// TIA Portal project "FinalYearProjectCode" (V17)
// This is the final combined plc code for the 5th year project

(* hardware
DEVICE "S7-1200 station_1"  S7-1200 Station
   slot 0: "Rack_0"  S7-1200 Rack  Rack  V1.0
   slot 1: "PLC_1"  CPU 1214C DC/DC/DC  6ES7 214-1AG40-0XB0  V4.2
   slot 2: "AI 4x13BIT/AQ 2x14BIT_1"  6ES7 234-4HE32-0XB0  V2.1
DEVICE "HMI_1"  TP700 Comfort
   slot 0: "HMI_1"  TP700 Comfort  6AV2 124-0GC01-0AX0  17.0.0.0
   slot 1: "HMI_RT_1"  TP700 Comfort  6AV2 124-0GC01-0AX0  17.0.0.0
   slot 5: "HMI_1.IE_CP_1"  PROFINET Interface  17.0.0.0
      slot 1: "PROFINET Interface_1"  PROFINET Interface
         slot 1: "Port_1"  Port
         slot 2: "Port_2"  Port
   slot 7: "HMI_1.MPI/DP_CP_1"  MPI/DP Interface  17.0.0.0
*)

// ===== PLC "PLC_1"  CPU 1214C DC/DC/DC =====

VAR_GLOBAL   // PLC tag table "Default tag table"
   "System_Byte" AT %MB100 : Byte;
   "FirstScan" AT %M100.0 : Bool;
   "DiagStatusUpdate" AT %M100.1 : Bool;
   "AlwaysTRUE" AT %M100.2 : Bool;
   "AlwaysFALSE" AT %M100.3 : Bool;
   "Clock_Byte" AT %MB101 : Byte;
   "Clock_10Hz" AT %M101.0 : Bool;
   "Clock_5Hz" AT %M101.1 : Bool;
   "Clock_2.5Hz" AT %M101.2 : Bool;
   "Clock_2Hz" AT %M101.3 : Bool;
   "Clock_1.25Hz" AT %M101.4 : Bool;
   "Clock_1Hz" AT %M101.5 : Bool;
   "Clock_0.625Hz" AT %M101.6 : Bool;
   "Clock_0.5Hz" AT %M101.7 : Bool;
END_VAR

VAR_GLOBAL   // PLC tag table "i_o_tags"
   "Voltage_transmitter" AT %IW96 : Int;
   "i_p_transducer" AT %QW96 : Int;
   "solar_sync" AT %Q0.1 : Bool;
   "compressor_rel" AT %Q0.2 : Bool;
   "caes_sync" AT %Q0.3 : Bool;
END_VAR

VAR_GLOBAL   // PLC tag table "HMI_tags"
   "HMI_START" AT %M0.0 : Bool;
   "HMI_STOP" AT %M0.1 : Bool;
   "Current_mode" AT %M0.2 : Bool;
END_VAR

VAR_GLOBAL   // PLC tag table "outMem_tags"
   "solarMainSync" AT %M1.0 : Bool;
   "solarStartSync" AT %M1.1 : Bool;
   "solarOnlySync" AT %M1.2 : Bool;
END_VAR

VAR_GLOBAL   // PLC tag table "caes_tags"
   "freq_feedback" AT %MD10 : Real;
   "first_in" AT %MD14 : Real;
   "i_p_mem1" AT %MW18 : Int;
   "controller_output" AT %MD20 : Real;
   "feedback_scale" AT %MD24 : Real;
   "control_scale" AT %MD28 : Real;
   "i_p_mem_2" AT %MW32 : Int;
   "press_mem" AT %MD34 : Real;
   "HMI_pressure" AT %MD38 : Real;
   "caesControlError" AT %MD42 : Real;
END_VAR

DATA_BLOCK "modbusConfig"   // DB3
{ S7_Optimized_Access := 'TRUE' }
VERSION : 0.1
   VAR
      MB_MODE : USInt;
      MB_DATA_ADDR_1 : UDInt := 30051;
      MB_DATA_ADDR_2 : UDInt := 30061;
      MB_DATA_ADDR_3 : UDInt := 30071;
      MB_DATA_ADDR_4 : UDInt := 30081;
      MB_DATA_ADDR_5 : UDInt := 30091;
      MB_DATA_LEN : UInt := 1;
      CONNECT_1 : TCON_IP_v4;
      CONNECT_2 : TCON_IP_v4;
      CONNECT_3 : TCON_IP_v4;
      CONNECT_4 : TCON_IP_v4;
      CONNECT_5 : TCON_IP_v4;
      STATUS_1 : Word;
      STATUS_2 : Word;
      STATUS_3 : Word;
      STATUS_4 : Word;
      STATUS_5 : Word;
      ERROR_1 : Bool;
      ERROR_2 : Bool;
      ERROR_3 : Bool;
      ERROR_4 : Bool;
      ERROR_5 : Bool;
   END_VAR
BEGIN
   CONNECT_1.InterfaceId := 64;
   CONNECT_1.ID := 1;
   CONNECT_1.ActiveEstablished := true;
   CONNECT_1.RemoteAddress.ADDR[1] := 172;
   CONNECT_1.RemoteAddress.ADDR[2] := 16;
   CONNECT_1.RemoteAddress.ADDR[3] := 41;
   CONNECT_1.RemoteAddress.ADDR[4] := 240;
   CONNECT_1.RemotePort := 502;
   CONNECT_2.InterfaceId := 64;
   CONNECT_2.ID := 2;
   CONNECT_2.ActiveEstablished := true;
   CONNECT_2.RemoteAddress.ADDR[1] := 172;
   CONNECT_2.RemoteAddress.ADDR[2] := 16;
   CONNECT_2.RemoteAddress.ADDR[3] := 41;
   CONNECT_2.RemoteAddress.ADDR[4] := 240;
   CONNECT_2.RemotePort := 502;
   CONNECT_3.InterfaceId := 64;
   CONNECT_3.ID := 3;
   CONNECT_3.ActiveEstablished := true;
   CONNECT_3.RemoteAddress.ADDR[1] := 172;
   CONNECT_3.RemoteAddress.ADDR[2] := 16;
   CONNECT_3.RemoteAddress.ADDR[3] := 41;
   CONNECT_3.RemoteAddress.ADDR[4] := 240;
   CONNECT_3.RemotePort := 502;
   CONNECT_4.InterfaceId := 64;
   CONNECT_4.ID := 4;
   CONNECT_4.ActiveEstablished := true;
   CONNECT_4.RemoteAddress.ADDR[1] := 172;
   CONNECT_4.RemoteAddress.ADDR[2] := 16;
   CONNECT_4.RemoteAddress.ADDR[3] := 41;
   CONNECT_4.RemoteAddress.ADDR[4] := 240;
   CONNECT_4.RemotePort := 502;
   CONNECT_5.InterfaceId := 64;
   CONNECT_5.ID := 5;
   CONNECT_5.ActiveEstablished := true;
   CONNECT_5.RemotePort := 502;
   CONNECT_5.RemoteAddress.ADDR[1] := 172;
   CONNECT_5.RemoteAddress.ADDR[2] := 16;
   CONNECT_5.RemoteAddress.ADDR[3] := 41;
   CONNECT_5.RemoteAddress.ADDR[4] := 240;
END_DATA_BLOCK

DATA_BLOCK "mbDataPTR"   // DB4
{ S7_Optimized_Access := 'FALSE' }
VERSION : 0.1
   VAR
      loadCurrent : Word;
      mainBusFreq : Word;
      solarSync : Word;
      solarFailsafe : Word;
      caesFailSafe : Word;
   END_VAR
BEGIN
END_DATA_BLOCK

FUNCTION "CAESControl" : Void   // FC1, LAD
{ S7_Optimized_Access := 'TRUE' }
VERSION : 0.1
BEGIN

REGION Network 1: Generator start_up
   // This block sets the generator
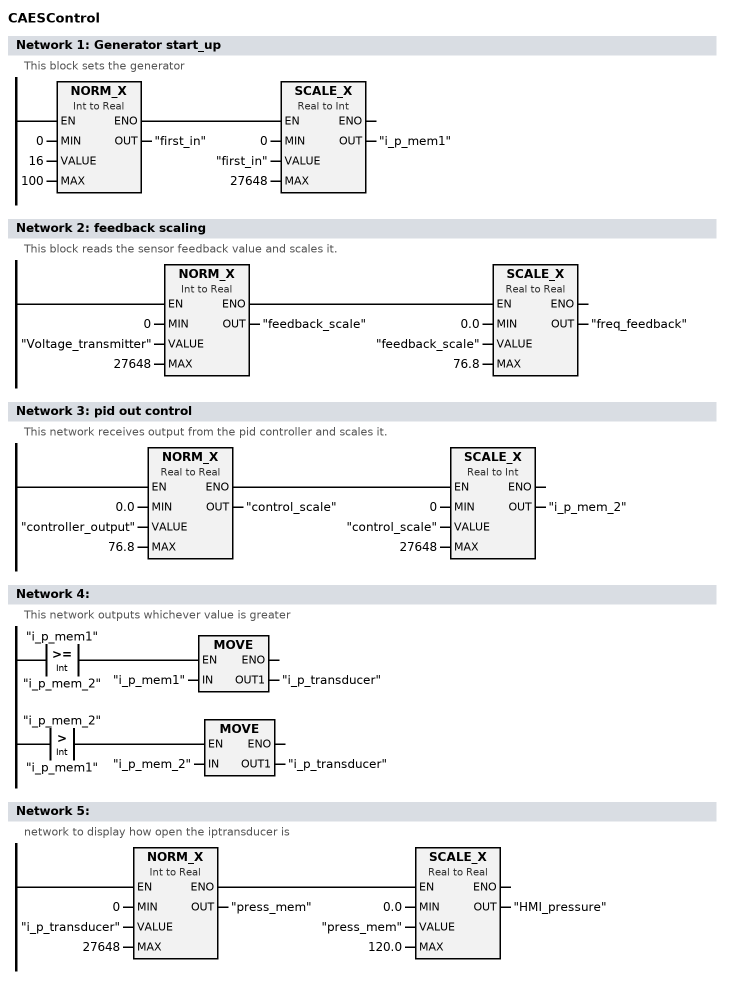
   RUNG wire#powerrail
      { S7_Templates := "[SrcType := Int, DestType := Real]" } Normalize(min := 0, value := 16, max := 100, out => "first_in")
      { S7_Templates := "[SrcType := Real, DestType := Int]" } Scale(min := 0, value := "first_in", max := 27648, out => "i_p_mem1")
   END_RUNG
   // the same network as SCL:
   "first_in" := NORM_X(MIN := 0, VALUE := 16, MAX := 100);
   "i_p_mem1" := SCALE_X(MIN := 0, VALUE := "first_in", MAX := 27648);
END_REGION

REGION Network 2: feedback scaling
   // This block reads the sensor feedback value and scales it.
   RUNG wire#powerrail
      { S7_Templates := "[SrcType := Int, DestType := Real]" } Normalize(min := 0, value := "Voltage_transmitter", max := 27648, out => "feedback_scale")
      { S7_Templates := "[SrcType := Real, DestType := Real]" } Scale(min := 0.0, value := "feedback_scale", max := 76.8, out => "freq_feedback")
   END_RUNG
   // the same network as SCL:
   "feedback_scale" := NORM_X(MIN := 0, VALUE := "Voltage_transmitter", MAX := 27648);
   "freq_feedback" := SCALE_X(MIN := 0.0, VALUE := "feedback_scale", MAX := 76.8);
END_REGION

REGION Network 3: pid out control
   // This network receives output from the pid controller and scales it.
   RUNG wire#powerrail
      { S7_Templates := "[SrcType := Real, DestType := Real]" } Normalize(min := 0.0, value := "controller_output", max := 76.8, out => "control_scale")
      { S7_Templates := "[SrcType := Real, DestType := Int]" } Scale(min := 0, value := "control_scale", max := 27648, out => "i_p_mem_2")
   END_RUNG
   // the same network as SCL:
   "control_scale" := NORM_X(MIN := 0.0, VALUE := "controller_output", MAX := 76.8);
   "i_p_mem_2" := SCALE_X(MIN := 0, VALUE := "control_scale", MAX := 27648);
END_REGION

REGION Network 4
   // This network outputs whichever value is greater
   RUNG wire#powerrail
      { S7_Templates := "SrcType := Int" } GE_Contact(in1 := "i_p_mem1", in2 := "i_p_mem_2")
      Move(in := "i_p_mem1", out1 => "i_p_transducer")
   END_RUNG
   RUNG wire#powerrail
      { S7_Templates := "SrcType := Int" } GT_Contact(in1 := "i_p_mem_2", in2 := "i_p_mem1")
      Move(in := "i_p_mem_2", out1 => "i_p_transducer")
   END_RUNG
   // the same network as SCL:
   IF "i_p_mem1" >= "i_p_mem_2" THEN "i_p_transducer" := "i_p_mem1"; END_IF;
   IF "i_p_mem_2" > "i_p_mem1" THEN "i_p_transducer" := "i_p_mem_2"; END_IF;
END_REGION

REGION Network 5
   // network to display how open the iptransducer is
   RUNG wire#powerrail
      { S7_Templates := "[SrcType := Int, DestType := Real]" } Normalize(min := 0, value := "i_p_transducer", max := 27648, out => "press_mem")
      { S7_Templates := "[SrcType := Real, DestType := Real]" } Scale(min := 0.0, value := "press_mem", max := 120.0, out => "HMI_pressure")
   END_RUNG
   // the same network as SCL:
   "press_mem" := NORM_X(MIN := 0, VALUE := "i_p_transducer", MAX := 27648);
   "HMI_pressure" := SCALE_X(MIN := 0.0, VALUE := "press_mem", MAX := 120.0);
END_REGION
END_FUNCTION

FUNCTION "comm" : Void   // FC2, LAD
{ S7_Optimized_Access := 'TRUE' }
VERSION : 0.1
BEGIN

REGION Network 1: Receive Load current
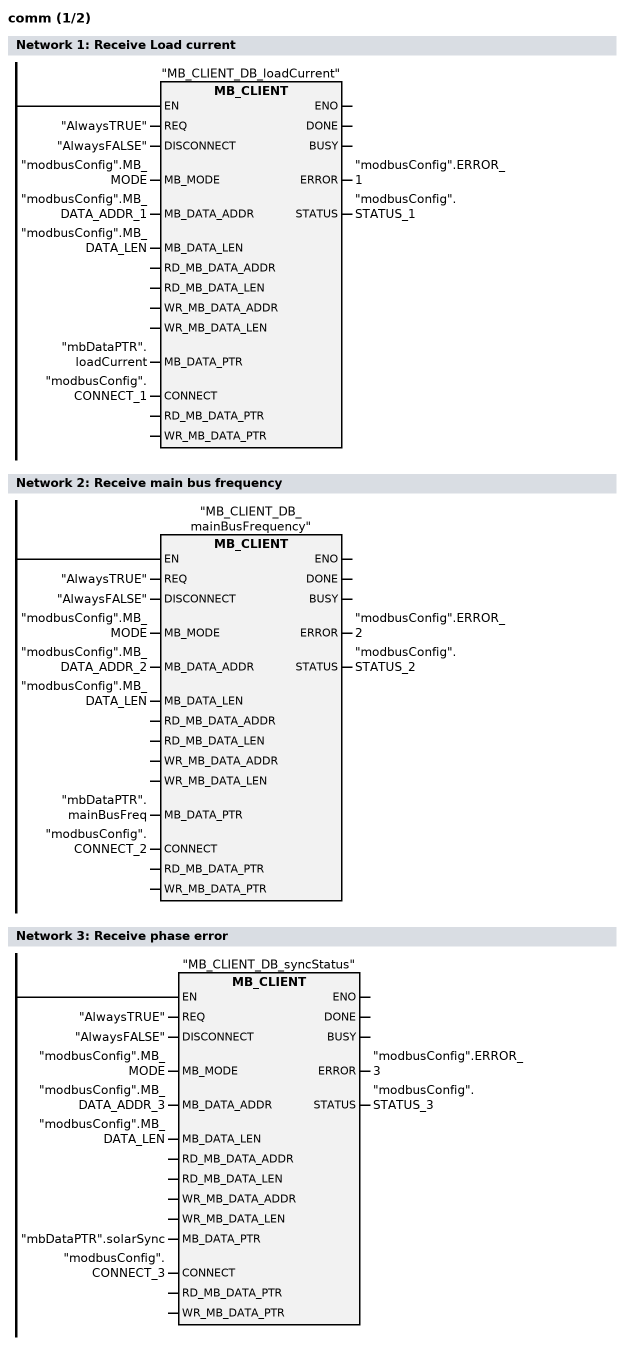
   "MB_CLIENT_DB_loadCurrent"(REQ := "AlwaysTRUE",   // MB_CLIENT
                           DISCONNECT := "AlwaysFALSE",
                           MB_MODE := "modbusConfig".MB_MODE,
                           MB_DATA_ADDR := "modbusConfig".MB_DATA_ADDR_1,
                           MB_DATA_LEN := "modbusConfig".MB_DATA_LEN,
                           MB_DATA_PTR := "mbDataPTR".loadCurrent,
                           CONNECT := "modbusConfig".CONNECT_1,
                           ERROR => "modbusConfig".ERROR_1,
                           STATUS => "modbusConfig".STATUS_1);
END_REGION

REGION Network 2: Receive main bus frequency
   "MB_CLIENT_DB_mainBusFrequency"(REQ := "AlwaysTRUE",   // MB_CLIENT
                           DISCONNECT := "AlwaysFALSE",
                           MB_MODE := "modbusConfig".MB_MODE,
                           MB_DATA_ADDR := "modbusConfig".MB_DATA_ADDR_2,
                           MB_DATA_LEN := "modbusConfig".MB_DATA_LEN,
                           MB_DATA_PTR := "mbDataPTR".mainBusFreq,
                           CONNECT := "modbusConfig".CONNECT_2,
                           ERROR => "modbusConfig".ERROR_2,
                           STATUS => "modbusConfig".STATUS_2);
END_REGION

REGION Network 3: Receive phase error
   "MB_CLIENT_DB_syncStatus"(REQ := "AlwaysTRUE",   // MB_CLIENT
                           DISCONNECT := "AlwaysFALSE",
                           MB_MODE := "modbusConfig".MB_MODE,
                           MB_DATA_ADDR := "modbusConfig".MB_DATA_ADDR_3,
                           MB_DATA_LEN := "modbusConfig".MB_DATA_LEN,
                           MB_DATA_PTR := "mbDataPTR".solarSync,
                           CONNECT := "modbusConfig".CONNECT_3,
                           ERROR => "modbusConfig".ERROR_3,
                           STATUS => "modbusConfig".STATUS_3);
END_REGION

REGION Network 4: Receive CAES Failsafe
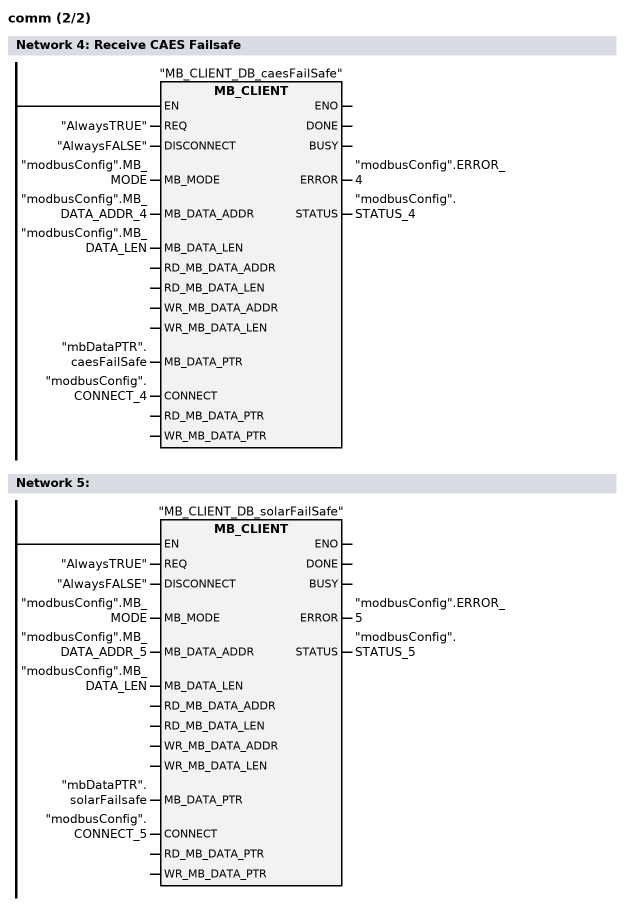
   "MB_CLIENT_DB_caesFailSafe"(REQ := "AlwaysTRUE",   // MB_CLIENT
                           DISCONNECT := "AlwaysFALSE",
                           MB_MODE := "modbusConfig".MB_MODE,
                           MB_DATA_ADDR := "modbusConfig".MB_DATA_ADDR_4,
                           MB_DATA_LEN := "modbusConfig".MB_DATA_LEN,
                           MB_DATA_PTR := "mbDataPTR".caesFailSafe,
                           CONNECT := "modbusConfig".CONNECT_4,
                           ERROR => "modbusConfig".ERROR_4,
                           STATUS => "modbusConfig".STATUS_4);
END_REGION

REGION Network 5
   "MB_CLIENT_DB_solarFailSafe"(REQ := "AlwaysTRUE",   // MB_CLIENT
                           DISCONNECT := "AlwaysFALSE",
                           MB_MODE := "modbusConfig".MB_MODE,
                           MB_DATA_ADDR := "modbusConfig".MB_DATA_ADDR_5,
                           MB_DATA_LEN := "modbusConfig".MB_DATA_LEN,
                           MB_DATA_PTR := "mbDataPTR".solarFailsafe,
                           CONNECT := "modbusConfig".CONNECT_5,
                           ERROR => "modbusConfig".ERROR_5,
                           STATUS => "modbusConfig".STATUS_5);
END_REGION
END_FUNCTION

FUNCTION "StopMode" : Void   // FC3, LAD
{ S7_Optimized_Access := 'TRUE' }
VERSION : 0.1
BEGIN

REGION Network 1
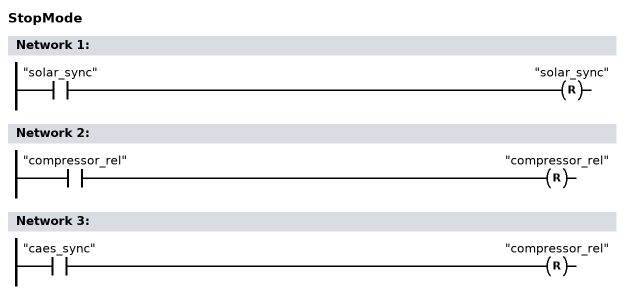
   RUNG wire#powerrail
      Contact( "solar_sync" )
      R_Coil( "solar_sync" )
   END_RUNG
   // the same network as SCL:
   IF "solar_sync" THEN "solar_sync" := FALSE; END_IF;
END_REGION

REGION Network 2
   RUNG wire#powerrail
      Contact( "compressor_rel" )
      R_Coil( "compressor_rel" )
   END_RUNG
   // the same network as SCL:
   IF "compressor_rel" THEN "compressor_rel" := FALSE; END_IF;
END_REGION

REGION Network 3
   RUNG wire#powerrail
      Contact( "caes_sync" )
      R_Coil( "compressor_rel" )
   END_RUNG
   // the same network as SCL:
   IF "caes_sync" THEN "compressor_rel" := FALSE; END_IF;
END_REGION
END_FUNCTION

FUNCTION "runMode" : Void   // FC4, LAD
{ S7_Optimized_Access := 'TRUE' }
VERSION : 0.1
BEGIN

REGION Network 1
   // This network controls the compressor socket
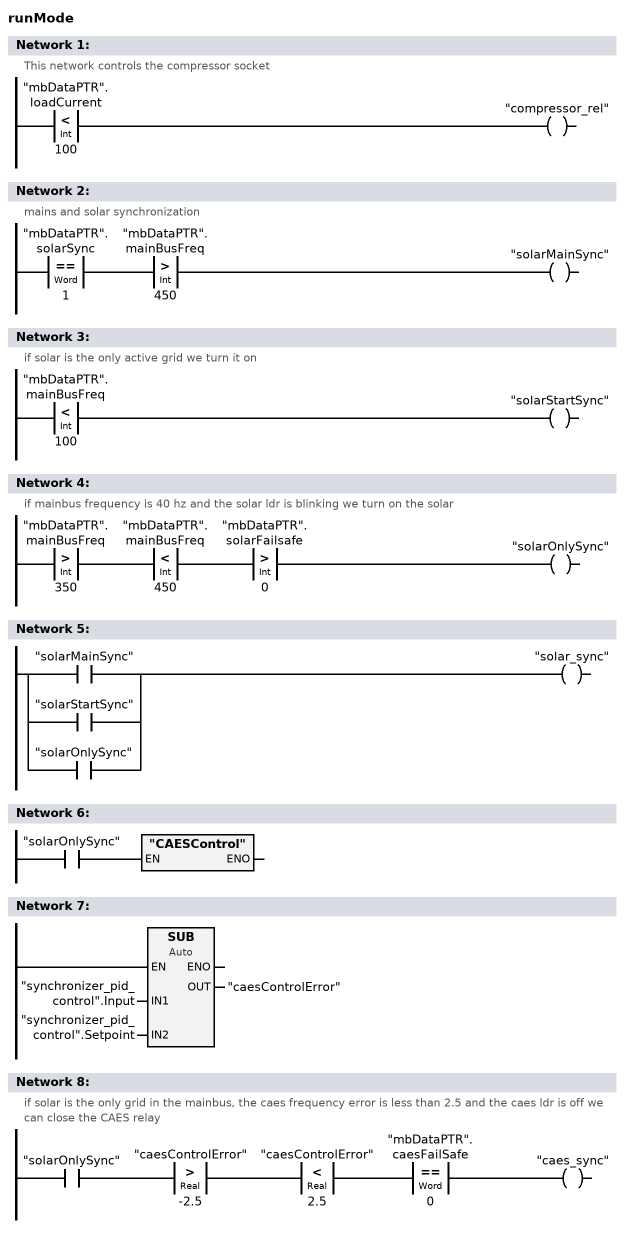
   RUNG wire#powerrail
      { S7_Templates := "SrcType := Int" } LT_Contact(in1 := "mbDataPTR".loadCurrent, in2 := 100)
      Coil( "compressor_rel" )
   END_RUNG
   // the same network as SCL:
   "compressor_rel" := "mbDataPTR".loadCurrent < 100;
END_REGION

REGION Network 2
   // mains and solar synchronization
   RUNG wire#powerrail
      { S7_Templates := "SrcType := Word" } EQ_Contact(in1 := "mbDataPTR".solarSync, in2 := 1)
      { S7_Templates := "SrcType := Int" } GT_Contact(in1 := "mbDataPTR".mainBusFreq, in2 := 450)
      Coil( "solarMainSync" )
   END_RUNG
   // the same network as SCL:
   "solarMainSync" := ("mbDataPTR".solarSync = 1) AND ("mbDataPTR".mainBusFreq > 450);
END_REGION

REGION Network 3
   // if solar is the only active grid we turn it on
   RUNG wire#powerrail
      { S7_Templates := "SrcType := Int" } LT_Contact(in1 := "mbDataPTR".mainBusFreq, in2 := 100)
      Coil( "solarStartSync" )
   END_RUNG
   // the same network as SCL:
   "solarStartSync" := "mbDataPTR".mainBusFreq < 100;
END_REGION

REGION Network 4
   // if mainbus frequency is 40 hz and the solar ldr is blinking we turn on the solar
   RUNG wire#powerrail
      { S7_Templates := "SrcType := Int" } GT_Contact(in1 := "mbDataPTR".mainBusFreq, in2 := 350)
      { S7_Templates := "SrcType := Int" } LT_Contact(in1 := "mbDataPTR".mainBusFreq, in2 := 450)
      { S7_Templates := "SrcType := Int" } GT_Contact(in1 := "mbDataPTR".solarFailsafe, in2 := 0)
      Coil( "solarOnlySync" )
   END_RUNG
   // the same network as SCL:
   "solarOnlySync" := ("mbDataPTR".mainBusFreq > 350) AND ("mbDataPTR".mainBusFreq < 450) AND ("mbDataPTR".solarFailsafe > 0);
END_REGION

REGION Network 5
   RUNG wire#powerrail
      Contact( "solarMainSync" )
      wire#w1
      Coil( "solar_sync" )
   END_RUNG
   RUNG wire#powerrail
      Contact( "solarStartSync" )
   END_RUNG wire#w1
   RUNG wire#powerrail
      Contact( "solarOnlySync" )
   END_RUNG wire#w1
   // the same network as SCL:
   "solar_sync" := "solarMainSync" OR "solarStartSync" OR "solarOnlySync";
END_REGION

REGION Network 6
   RUNG wire#powerrail
      Contact( "solarOnlySync" )
      "CAESControl"()
   END_RUNG
   // the same network as SCL:
   IF "solarOnlySync" THEN "CAESControl"(); END_IF;
END_REGION

REGION Network 7
   RUNG wire#powerrail
      Sub(in1 := "synchronizer_pid_control".Input, in2 := "synchronizer_pid_control".Setpoint, out => "caesControlError")
   END_RUNG
   // the same network as SCL:
   "caesControlError" := "synchronizer_pid_control".Input - "synchronizer_pid_control".Setpoint;
END_REGION

REGION Network 8
   // if solar is the only grid in the mainbus, the caes frequency error is less than 2.5 and the caes ldr is off we can close the CAES relay
   RUNG wire#powerrail
      Contact( "solarOnlySync" )
      { S7_Templates := "SrcType := Real" } GT_Contact(in1 := "caesControlError", in2 := -2.5)
      { S7_Templates := "SrcType := Real" } LT_Contact(in1 := "caesControlError", in2 := 2.5)
      { S7_Templates := "SrcType := Word" } EQ_Contact(in1 := "mbDataPTR".caesFailSafe, in2 := 0)
      Coil( "caes_sync" )
   END_RUNG
   // the same network as SCL:
   "caes_sync" := "solarOnlySync" AND ("caesControlError" > (-2.5)) AND ("caesControlError" < 2.5) AND ("mbDataPTR".caesFailSafe = 0);
END_REGION
END_FUNCTION

ORGANIZATION_BLOCK "Main"   // OB1, LAD, ProgramCycle
TITLE = "Main Program Sweep (Cycle)"
{ S7_Optimized_Access := 'TRUE' }
VERSION : 0.1
   VAR_INPUT
      Initial_Call : Bool;   // Initial call of this OB
      Remanence : Bool;   // =True, if remanent data are available
   END_VAR
BEGIN

REGION Network 1
   // this calls the CAES control circuit
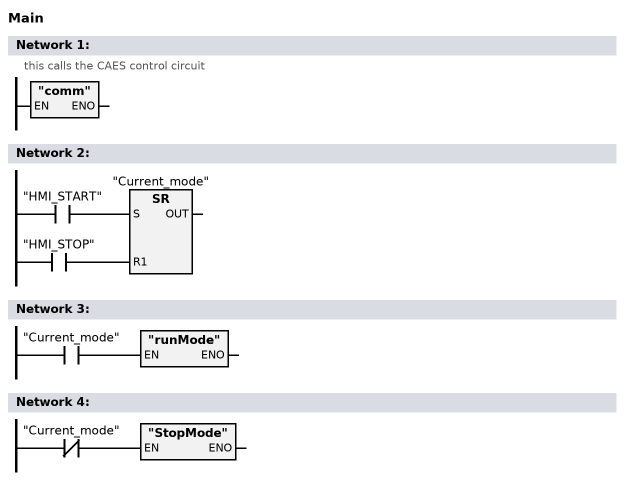
   RUNG wire#powerrail
      "comm"()
   END_RUNG
   // the same network as SCL:
   "comm"();
END_REGION

REGION Network 2
   RUNG wire#powerrail
      Contact( "HMI_START" )
      S_SR(operand := "Current_mode", r1 := wire#w1)
   END_RUNG
   RUNG wire#powerrail
      Contact( "HMI_STOP" )
   END_RUNG wire#w1
   // the same network as SCL:
   IF "HMI_START" THEN
       "Current_mode" := TRUE;   // SR flip-flop
   END_IF;
   IF "HMI_STOP" THEN "Current_mode" := FALSE; END_IF;
END_REGION

REGION Network 3
   RUNG wire#powerrail
      Contact( "Current_mode" )
      "runMode"()
   END_RUNG
   // the same network as SCL:
   IF "Current_mode" THEN "runMode"(); END_IF;
END_REGION

REGION Network 4
   RUNG wire#powerrail
      I_Contact( "Current_mode" )
      "StopMode"()
   END_RUNG
   // the same network as SCL:
   IF NOT "Current_mode" THEN "StopMode"(); END_IF;
END_REGION
END_ORGANIZATION_BLOCK

ORGANIZATION_BLOCK "Cyclic interrupt"   // OB30, LAD, CyclicInterrupt
{ S7_Optimized_Access := 'TRUE' }
VERSION : 0.1
   VAR_INPUT
      Initial_Call : Bool;   // Initial call of this OB
      Event_Count : Int;   // Events discarded
   END_VAR
BEGIN

REGION Network 1
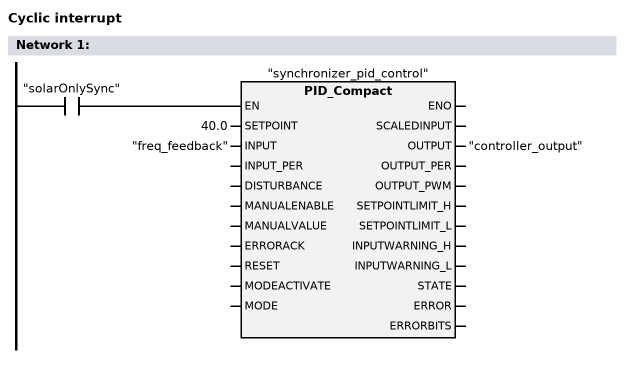
   IF "solarOnlySync" THEN
       "synchronizer_pid_control"(Setpoint := 40.0, Input := "freq_feedback", Output => "controller_output");   // PID_Compact
   END_IF;
END_REGION
END_ORGANIZATION_BLOCK

(* ===== HMI "HMI_RT_1" =====
system functions are stored by id; their names below are inferred from use
connection "HMI_Connection_1": ETHERNET, S7_1200_OMS

HMI tags "Default tag table"
   "synchronizer_pid_control_Output" : Real = PLC synchronizer_pid_control.Output, 1 s
   "synchronizer_pid_control_Input" : Real = PLC synchronizer_pid_control.Input, 1 s
   "synchronizer_pid_control_Setpoint" : Real = PLC synchronizer_pid_control.Setpoint, 1 s
   "synchronizer_pid_control_CtrlParamsBackUp_Gain" : Real = PLC synchronizer_pid_control.CtrlParamsBackUp.Gain, 1 s
   "synchronizer_pid_control_CtrlParamsBackUp_Ti" : Real = PLC synchronizer_pid_control.CtrlParamsBackUp.Ti, 1 s
   "synchronizer_pid_control_CtrlParamsBackUp_Td" : Real = PLC synchronizer_pid_control.CtrlParamsBackUp.Td, 1 s
   "HMI_pressure" : Real = PLC HMI_pressure AT %MD38, 1 s
   "mbDataPTR_loadCurrent" : Word = PLC mbDataPTR.loadCurrent AT %DB4.DBW0, 1 s
   "mbDataPTR_mainBusFreq" : Word = PLC mbDataPTR.mainBusFreq AT %DB4.DBW2, 1 s
   "mbDataPTR_solarSync" : Word = PLC mbDataPTR.solarSync AT %DB4.DBW4, 1 s
   "mbDataPTR_caesFailSafe" : Word = PLC mbDataPTR.caesFailSafe AT %DB4.DBW8, 1 s
   "mbDataPTR_solarFailsafe" : Word = PLC mbDataPTR.solarFailsafe AT %DB4.DBW6, 1 s
   "HMI_START" : Bool = PLC HMI_START AT %M0.0, 1 s
   "HMI_STOP" : Bool = PLC HMI_STOP AT %M0.1, 1 s

screen "CAES_PID" 800x480
   TrendView "Trend view_1" at 3,41 size 594x437
   TextField "Text field_1" at 151,8 size 543x34; Text 'CAES PID CONTROLLER VISUALIZATION'
   IOField "I/O field_1" at 699,43 size 96x32; FormatPattern 99.999
      ProcessValue <- "synchronizer_pid_control_CtrlParamsBackUp_Gain"
   IOField "I/O field_2" at 700,86 size 96x32; FormatPattern 99.999
      ProcessValue <- "synchronizer_pid_control_CtrlParamsBackUp_Ti"
   IOField "I/O field_3" at 700,130 size 96x32; FormatPattern 99.999
      ProcessValue <- "synchronizer_pid_control_CtrlParamsBackUp_Td"
   TextField "Text field_2" at 658,43 size 36x31; Text 'Kp'
   TextField "Text field_3" at 657,86 size 29x31; Text 'Ki'
   TextField "Text field_4" at 656,129 size 36x31; Text 'Kd'
   Gauge "Gauge_1" at 598,264 size 200x200; CaptionText 'CAES pressure'; UnitText 'psi'
      ProcessValue <- "HMI_pressure"
   TextField "Text field_5" at 667,227 size 60x31; Text 'Pout'
   Button "Button_1" at 22,8 size 96x32; TextOff 'HOME'
      on Press: ActivateScreen("HOME", 0)

screen "HOME" 800x480
   Button "Button_1" at 18,16 size 96x32; TextOff 'CAES'
      on Press: ActivateScreen("CAES_PID", 0)
   TextField "Text field_1" at 52,87 size 147x23; Text 'LOAD CURRENT'
   TextField "Text field_2" at 52,126 size 210x23; Text 'MAIN BUS FREQUENCY'
   TextField "Text field_3" at 52,165 size 197x23; Text 'SOLAR SYNC STATUS'
   TextField "Text field_4" at 52,204 size 209x23; Text 'CAES FAILSAFE VALUE'
   TextField "Text field_5" at 53,243 size 222x23; Text 'SOLAR FAILSAFE VALUE'
   IOField "I/O field_1" at 287,78 size 96x32; FormatPattern 99999
      ProcessValue <- "mbDataPTR_loadCurrent"
   IOField "I/O field_2" at 287,122 size 96x32; FormatPattern 99999
      ProcessValue <- "mbDataPTR_mainBusFreq"
   IOField "I/O field_3" at 286,162 size 96x32; FormatPattern 99999
      ProcessValue <- "mbDataPTR_solarSync"
   IOField "I/O field_4" at 285,202 size 96x32; FormatPattern 99999
      ProcessValue <- "mbDataPTR_caesFailSafe"
   IOField "I/O field_5" at 284,242 size 96x32; FormatPattern 99999
      ProcessValue <- "mbDataPTR_solarFailsafe"
   Button "Button_2" at 37,342 size 96x32; TextOff 'START'
      on Press: SetBit("HMI_START")
      on Release: ResetBit("HMI_START")
   Button "Button_3" at 286,342 size 96x32; TextOff 'STOP'
      on Press: SetBit("HMI_STOP")
      on Release: ResetBit("HMI_STOP")
   TextField "Text field_6" at 621,109 size 97x23; Text 'WIZARDS'
   TextField "Text field_7" at 656,149 size 28x23; Text 'OF'
   TextField "Text field_8" at 664,205 size 47x23; Text 'THE'
   TextField "Text field_9" at 629,253 size 52x23; Text 'GRID'
*)